INTERFACE ITF_Error

PROPERTY pAckError : BOOL
GET
END_GET
SET
END_SET
END_PROPERTY

PROPERTY pError : BOOL
GET
END_GET
SET
END_SET
END_PROPERTY

PROPERTY pErrorCode : udint
GET
END_GET
SET
END_SET
END_PROPERTY

PROPERTY pErrorDescription : T_MaxString
GET
END_GET
SET
END_SET
END_PROPERTY

END_INTERFACE

(* stored: Version 1.1.0.1, ProductVersion 3.1.4024.12
   Itf ITF_Error: Id {5a56ba58-d4fe-0c79-372c-3dcfc76b6fd4}
   Property pAckError: Id {4105a70e-ef46-02e5-3e9a-6c5613957bf3}
   Get Get: Id {c57bea28-f8a0-07ec-1924-bb3c9119f45a}
   Set Set: Id {15dd27b6-ad00-0fce-0e53-a6af85408f92}
   Property pError: Id {9b55ee16-8489-022b-3f94-208e2a04a549}
   Get Get: Id {7846a499-8690-0aa6-0ed1-b25710f6f7e6}
   Set Set: Id {6ecd69c2-6fa9-0453-2cba-eaf6d10fc275}
   Property pErrorCode: Id {83dab1d4-4699-0a08-0652-15adbb33cf23}
   Get Get: Id {d4285aaa-37e4-07cb-18e2-cf05d2029a55}
   Set Set: Id {7e8c8cee-3ebb-0408-06be-a71ce8342521}
   Property pErrorDescription: Id {4b340105-ef65-07bf-10dc-0503155ae2fe}
   Get Get: Id {d29cce07-4303-0606-248b-dae467ec173e}
   Set Set: Id {50dac819-e7c6-0af3-1f2c-4f22fec71e45} *)
